	// Error
	E_SA_POS_SM_STATE.ERROR:
		IF ch_ctrl.nCmd = E_SA_CH_CMD.CALIB	THEN
			ch_ctrl.nCmd 			:= E_SA_CH_CMD.NONE;	// Reset command
			stat.nPosState 		:= E_SA_POS_SM_STATE.CALIB;
			stat.bInitialised	:= FALSE;
			stat.sStatus		:= 'Calibrating...';
			M_SetState(E_SA_POS_ELT_STATE.NOTOP);
			M_SetSubstate(E_SA_POS_ELT_SUBSTATE.NOTOP_NOTREADY);
			M_SetNextPosState	:= TRUE;	// State HAS changed
		ELSIF ch_ctrl.nCmd = E_SA_CH_CMD.REF	THEN
			ch_ctrl.nCmd 			:= E_SA_CH_CMD.NONE;	// Reset command
			stat.nPosState 		:= E_SA_POS_SM_STATE.INIT;
			stat.bInitialised	:= FALSE;
			stat.sStatus		:= 'Referencing/INIT Started';
			M_SetState(E_SA_POS_ELT_STATE.NOTOP);
			M_SetSubstate(E_SA_POS_ELT_SUBSTATE.NOTOP_NOTREADY);
			M_SetNextPosState	:= TRUE;	// State HAS changed
		ELSIF ch_ctrl.nCmd = E_SA_CH_CMD.MOV	THEN
			ch_ctrl.nCmd 			:= E_SA_CH_CMD.NONE;	// Reset command
			stat.stState.bACTIVELY_MOVING	:= TRUE;
			stat.stState.bIN_POSITION		:= FALSE;
			stat.nPosState 		:= E_SA_POS_SM_STATE.MOVING;
			stat.nLastPosState 	:= E_SA_POS_SM_STATE.OP;
			stat.sStatus		:= 'Moving...';
			M_SetSubstate(E_SA_POS_ELT_SUBSTATE.OP_MOVING);
			M_SetNextPosState	:= TRUE;	// State HAS changed
		ELSIF ch_ctrl.nCmd = E_SA_CH_CMD.RESET	THEN
			ch_ctrl.nCmd 			:= E_SA_CH_CMD.NONE;	// Reset command
			stat.nPosState 		:= E_SA_POS_SM_STATE.NOT_READY;
			stat.bInitialised	:= FALSE;
			//stat.nErrorCode		:= E_SA_CH_ERROR.OK;
			stat.nErrorCode		:= E_SM_ERROR.OK; 
			stat.sErrorText		:= 'OK';
			stat.sStatus		:= 'Positioner Reset';
			M_SetState(E_SA_POS_ELT_STATE.NOTOP);
			M_SetSubstate(E_SA_POS_ELT_SUBSTATE.NOTOP_NOTREADY);
			M_SetNextPosState	:= TRUE;	// State HAS changed
		ELSE
			stat.sStatus		:= M_GetErrorString();
			M_SetNextPosState	:= FALSE;	// State has NOT changed
		END_IF
END_CASE

*)
END_METHOD

METHOD M_SetState
VAR_INPUT
	nState: E_SA_POS_ELT_STATE;
	//nState: E_RS_BASE_STATE;
END_VAR
stat.nState	:= nState;

// Set substate string
CASE nState	OF
	E_SA_POS_ELT_STATE.NOTOP: 	stat.sState	:= 'NOT OP';
	E_SA_POS_ELT_STATE.OP: 		stat.sState	:= 'OPERATIONAL';
END_CASE
END_METHOD

METHOD M_SetSubstate
VAR_INPUT
	nSubstate: E_SA_POS_ELT_SUBSTATE;
	//nSubstate: E_RS_BASE_SUBSTATE;
END_VAR
stat.nSubstate	:= nSubstate;

// Set substate string
CASE nSubstate	OF
	E_SA_POS_ELT_SUBSTATE.NOTOP_NOTREADY: 		
		stat.sSubstate	:= 'NOT READY';
		stat.sStatus	:= '';
	E_SA_POS_ELT_SUBSTATE.NOTOP_READY: 			stat.sSubstate	:= 'READY';
	E_SA_POS_ELT_SUBSTATE.NOTOP_INITIALIZING:	stat.sSubstate	:= 'INITIALIZING';
	E_SA_POS_ELT_SUBSTATE.NOTOP_ABORTING:		stat.sSubstate	:= 'ABORTING';
	E_SA_POS_ELT_SUBSTATE.NOTOP_ERROR:			stat.sSubstate	:= 'ERROR';
	
	E_SA_POS_ELT_SUBSTATE.OP_STANDSTILL:		stat.sSubstate	:= 'STANDSTILL';            
	E_SA_POS_ELT_SUBSTATE.OP_MOVING:			stat.sSubstate	:= 'MOVING';
	E_SA_POS_ELT_SUBSTATE.OP_SETTING_POS:		stat.sSubstate	:= 'SETTING POS';
	E_SA_POS_ELT_SUBSTATE.OP_STOPPING:			stat.sSubstate	:= 'STOPPING';
	E_SA_POS_ELT_SUBSTATE.OP_ERROR:				stat.sSubstate	:= 'ERROR';
	
END_CASE
END_METHOD

//
// Convert Positioner status from Device to User mode.
//
METHOD M_UpdateStatus
VAR_INPUT
END_VAR
//
// Update bEnabled flag.
// If TRUE, it means that the amplifier is enabled and the sensor is present.
//
//stat.bEnabled	:= stat.stState.bAMPLIFIER_ENABLED AND  stat.stState.bSENSOR_PRESENT;


//
// Set the in-position flag
//
//stat.bInPosition	:= stat.stState.bIN_POSITION;


//
// Set target and actual positions in [UU]
//

//stat.lrPosTarget	:= M_ConvertPosDev2User(stat.devStatus.lnPosTarget);
//stat.lrPosActual	:= M_ConvertPosDev2User(stat.devStatus.lnPosActual);


//
// Set Standard ELT States and Substates
//


//
// Substate
//
CASE stat.nState OF
	E_SA_POS_ELT_STATE.NOTOP:
	/////////////////////////
	IF stat.bError	THEN
		M_SetSubstate(E_SA_POS_ELT_SUBSTATE.NOTOP_ERROR);
	ELSIF	stat.nPosState = E_SA_POS_SM_STATE.NOT_READY	THEN
		M_SetSubstate(E_SA_POS_ELT_SUBSTATE.NOTOP_NOTREADY);
	ELSIF 	stat.nPosState = E_SA_POS_SM_STATE.CALIB  		OR
			stat.nPosState = E_SA_POS_SM_STATE.INIT  		OR
			stat.nPosState = E_SA_POS_SM_STATE.POST_INIT	OR	
			stat.nPosState = E_SA_POS_SM_STATE.CALIB_REF  		THEN
		M_SetSubstate(E_SA_POS_ELT_SUBSTATE.NOTOP_INITIALIZING);
	ELSIF 	stat.nPosState = E_SA_POS_SM_STATE.READY  	THEN
		M_SetSubstate(E_SA_POS_ELT_SUBSTATE.NOTOP_READY);
	ELSE
		M_SetSubstate(E_SA_POS_ELT_SUBSTATE.NOTOP_NOTREADY);
	END_IF
	
	E_SA_POS_ELT_STATE.OP:
	//////////////////////
	IF stat.stState.bACTIVELY_MOVING	THEN
		IF stat.nPosState = E_SA_POS_SM_STATE.STOP	THEN
			M_SetSubstate(E_SA_POS_ELT_SUBSTATE.OP_STOPPING);
		ELSE
			M_SetSubstate(E_SA_POS_ELT_SUBSTATE.OP_MOVING);
		END_IF
	ELSIF stat.stState.bERROR	THEN
		M_SetSubstate(E_SA_POS_ELT_SUBSTATE.OP_ERROR);
	ELSE
		M_SetSubstate(E_SA_POS_ELT_SUBSTATE.OP_STANDSTILL);
	END_IF
END_CASE
END_METHOD

{attribute 'TcRpcEnable':='1'}
{attribute 'TcRpcEnable'}
METHOD RPC_MoveToFilterPosition : INT
VAR_INPUT
	in_nFilterPos:		DINT;	// 1 - 6
	
END_VAR

// If the SmarAct MCS2 Controller is in error,
// the positioner cannot be controlled.
//IF stat.nCtrlErrorCode <> 0  OR  stat.nCtrlState <> E_RS_BASE_STATE.OP THEN
//	RPC_MoveToFilterPosition	:= M_SetRpcStatus(E_SA_RPC_ERROR.CTRL_ERROR);
//	RETURN;
//END_IF


// RPC calls are not allowed in Local mode.
IF stat.bLocal THEN
	RPC_MoveToFilterPosition	:= M_SetRpcStatus(E_SA_RPC_ERROR.LOCAL);
	RETURN;
// Move Absolute command is accepted only in OP state.
ELSIF	stat.nState <> E_SA_POS_ELT_STATE.OP	THEN
	RPC_MoveToFilterPosition	:= M_SetRpcStatus(E_SA_RPC_ERROR.NOT_OP);
	RETURN;
// The positioner has to be initialised / OP (operational), i.e. already REFerenced.
ELSIF	NOT stat.bInitialised	THEN
	RPC_MoveToFilterPosition	:= M_SetRpcStatus(E_SA_RPC_ERROR.CH_NOT_OP);
	RETURN;

// If SW limits are active, check the limits
ELSIF in_nFilterPos > 6  THEN 	
		RPC_MoveToFilterPosition	:= M_SetRpcStatus(E_SA_RPC_ERROR.SW_LIMIT_UPPER);
		RETURN;
ELSIF in_nFilterPos < 1  THEN 	
		RPC_MoveToFilterPosition	:= M_SetRpcStatus(E_SA_RPC_ERROR.SW_LIMIT_LOWER);
		RETURN;
	
END_IF

// Set command
ch_ctrl.nCmd	:= E_SA_CH_CMD.MOV;
ch_ctrl.lrPos	:= in_nFilterPos;



// Call was successful
RPC_MoveToFilterPosition	:= M_SetRpcStatus(E_SA_RPC_ERROR.OK);
END_METHOD

END_FUNCTION_BLOCK

// ---- GlobalTextList.TcGTLO
TEXTLIST GlobalTextList
  14 = '%.2f'
  229 = '%.4f'
  992 = '%.5f'
  28 = '%.6f'
  860 = '%.7f'
  360 = '%s'
  753 = 'Absolute position used by "MOVE ABS"'
  174 = 'Backlash'
  107 = 'GREEN if initialised'
  963 = 'INIT'
  701 = 'Last Command'
  1168 = 'Offset (REL)'
  1376 = 'Position (ABS)'
  510 = 'Position Difference'
  2351 = 'Relative offset used by "MOVE REL"'
  1111 = 'Speed (Pos)'
  1135 = 'Speed (Vel)'
  1119 = 'Target              Actual'
  960 = 'Target           Actual'
END_TEXTLIST

// ---- VISUs/DL_Servo_1_Config.TcVIS
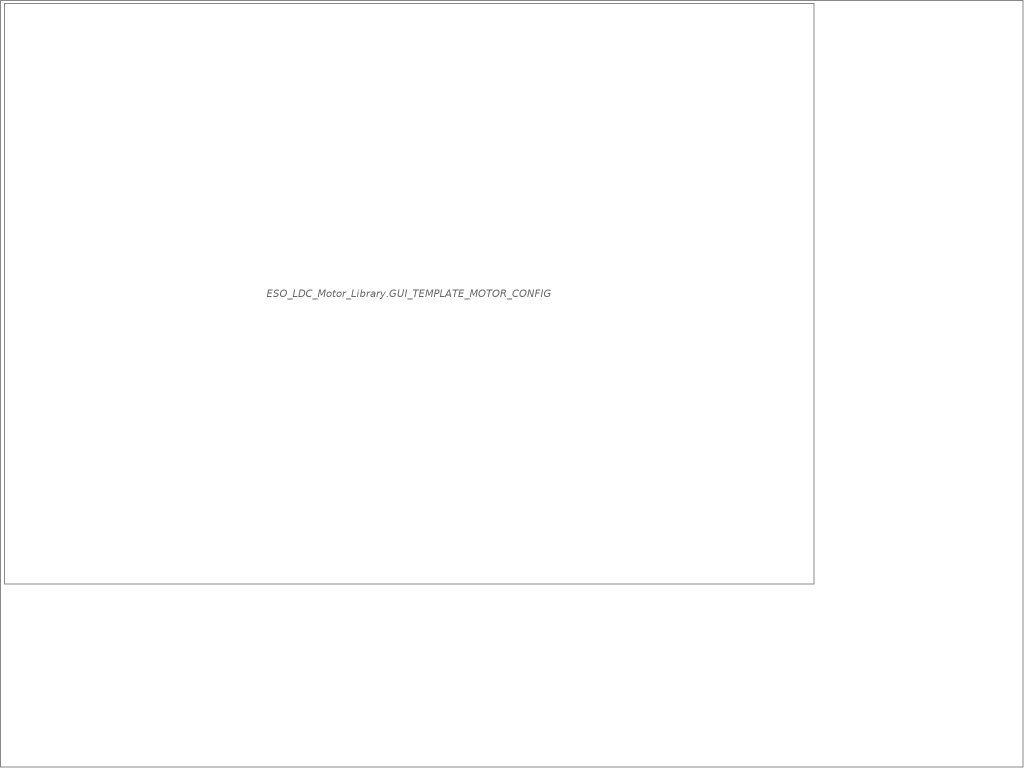
VISUALIZATION DL_Servo_1_Config  // 1024x768
    Frame (4,3 810x581)
        shows ESO_LDC_Motor_Library.GUI_TEMPLATE_MOTOR_CONFIG(m_Instance := MAIN.DL_Servo_1)
END_VISUALIZATION

// ---- VISUs/DL_Servo_1_Control.TcVIS
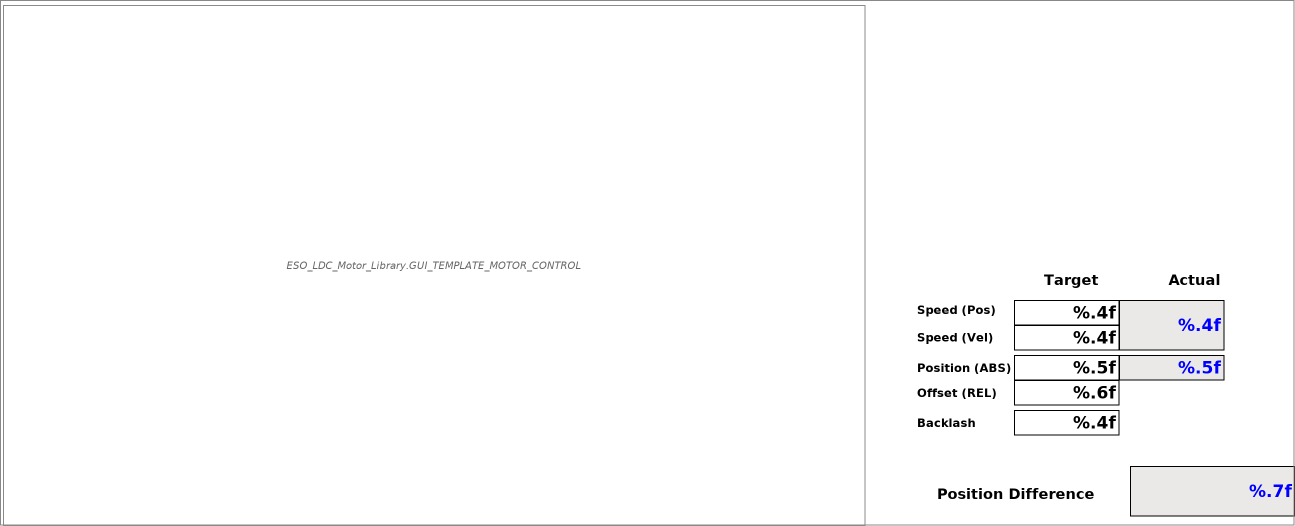
VISUALIZATION DL_Servo_1_Control  // 1295x526
    Frame (3,5 862x521)
        shows ESO_LDC_Motor_Library.GUI_TEMPLATE_MOTOR_CONTROL(m_Instance := MAIN.DL_Servo_1)
    Rectangle (914,300 95x20), "Speed (Pos)"
    Rectangle (1119,355 105x25), "%.5f", text variable: MAIN.DL_Servo_1.stat.lrPosActual, input disabled if: false
    Rectangle (1041,270 190x20), "Target Actual"
    Rectangle (914,358 95x20), "Position (ABS)"
    Rectangle (1119,300 105x50), "%.4f", text variable: MAIN.DL_Servo_1.stat.lrVelActual, input disabled if: false
    Rectangle (1014,325 105x25), "%.4f", text variable: MAIN.DL_Servo_1.ctrl.lrVelocity
        OnMouseDown: write the text variable via Default
    Rectangle (914,413 95x20), "Backlash"
    Rectangle (1014,410 105x25), "%.4f", text variable: MAIN.DL_Servo_1.cfg.lrBacklash
        OnMouseDown: write the text variable via Default
    Rectangle (914,325 95x25), "Speed (Vel)"
    Rectangle (1014,355 105x25), "%.5f", tooltip "Absolute position used by "MOVE ABS"", text variable: MAIN.DL_Servo_1.ctrl.lrPosition
        OnMouseDown: write the text variable via Default
    Rectangle (1014,300 105x25), "%.4f", text variable: MAIN.DL_Servo_1.cfg.lrDefaultVelocity
        OnMouseDown: write the text variable via Default
    Rectangle (914,383 95x20), "Offset (REL)"
    Rectangle (1014,380 105x25), "%.6f", tooltip "Relative offset used by "MOVE REL"", text variable: MAIN.DL_Servo_1.ctrl.lrOffset
        OnMouseDown: write the text variable via Default
    Rectangle (1130,466 165x50), "%.7f", text variable: MAIN.DL_Servo_1.stat.lrPosError, input disabled if: false
    Rectangle (934,484 190x20), "Position Difference"
END_VISUALIZATION

// ---- VISUs/Filter_Wheel.TcVIS
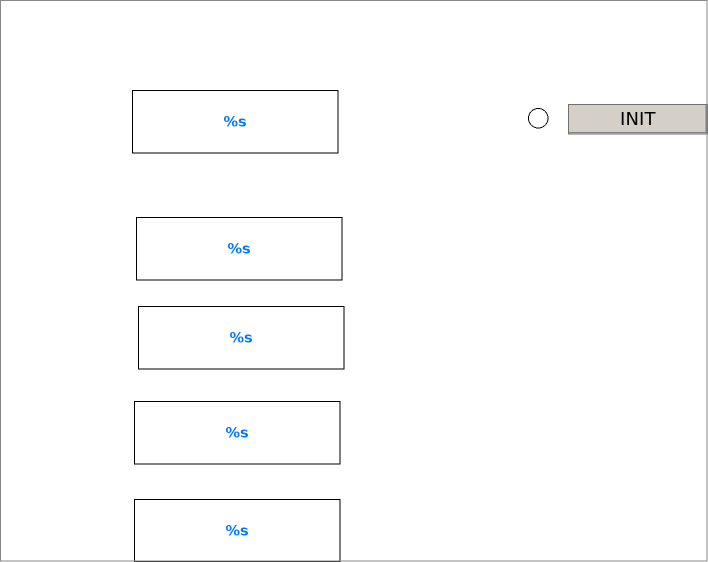
VISUALIZATION Filter_Wheel  // 708x562
    Rectangle (132,90 206x63), "%s", tooltip "Last Command", text variable: MAIN.FILTER_WHEEL.stat.sReply
    Rectangle (136,217 206x63), "%s", tooltip "Last Command", text variable: MAIN.FILTER_WHEEL.stat.sDeviceID
    Rectangle (138,306 206x63), "%s", tooltip "Last Command", text variable: MAIN.FILTER_WHEEL.stat.nCurrentFilterPosition
    Rectangle (134,401 206x63), "%s", tooltip "Last Command", text variable: MAIN.FILTER_WHEEL.stat.sFilterPosition
    Rectangle (134,499 206x63), "%s", tooltip "Last Command", text variable: MAIN.FILTER_WHEEL.stat.bMoveSpeed
    Button (568,104 140x30), "INIT"
        OnMouseClick: execute { MAIN.FILTER_WHEEL.ch_ctrl.nCmd:=E_SA_CH_CMD.REF; }
    Ellipse (528,108 20x20), tooltip "GREEN if initialised", colour toggle: MAIN.FILTER_WHEEL.stat.bInitialised
END_VISUALIZATION

// ---- VISUs/GUI_DL_2.TcVIS
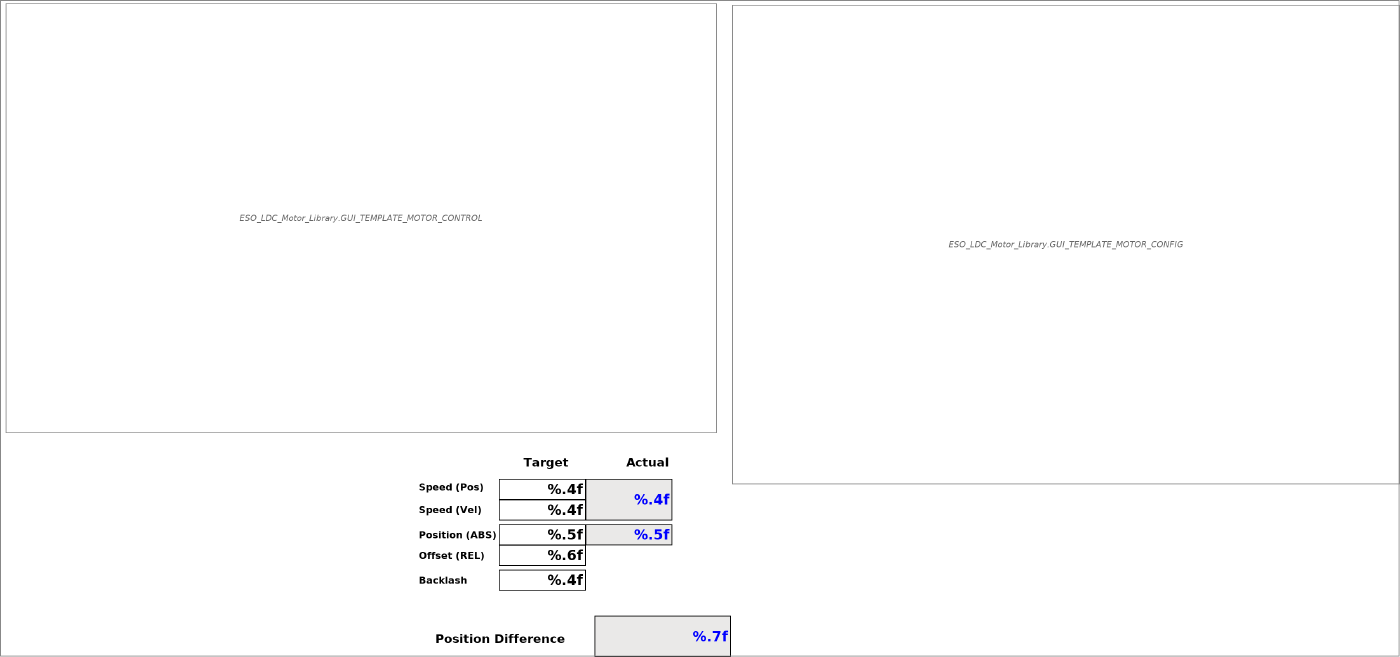
VISUALIZATION GUI_DL_2  // 1698x797
    Frame (7,4 862x521)
        shows ESO_LDC_Motor_Library.GUI_TEMPLATE_MOTOR_CONTROL(m_Instance := MAIN.DL_2)
    Frame (888,6 810x581)
        shows ESO_LDC_Motor_Library.GUI_TEMPLATE_MOTOR_CONFIG(m_Instance := MAIN.DL_2)
    Rectangle (505,581 95x20), "Speed (Pos)"
    Rectangle (710,636 105x25), "%.5f", text variable: MAIN.DL_2.stat.lrPosActual, input disabled if: false
    Rectangle (632,551 190x20), "Target Actual"
    Rectangle (505,639 95x20), "Position (ABS)"
    Rectangle (710,581 105x50), "%.4f", text variable: MAIN.DL_2.stat.lrVelActual, input disabled if: false
    Rectangle (605,606 105x25), "%.4f", text variable: MAIN.DL_2.ctrl.lrVelocity
        OnMouseDown: write the text variable via Default
    Rectangle (505,694 95x20), "Backlash"
    Rectangle (605,691 105x25), "%.4f", text variable: MAIN.DL_2.cfg.lrBacklash
        OnMouseDown: write the text variable via Default
    Rectangle (505,606 95x25), "Speed (Vel)"
    Rectangle (605,636 105x25), "%.5f", tooltip "Absolute position used by "MOVE ABS"", text variable: MAIN.DL_2.ctrl.lrPosition
        OnMouseDown: write the text variable via Default
    Rectangle (605,581 105x25), "%.4f", text variable: MAIN.DL_2.cfg.lrDefaultVelocity
        OnMouseDown: write the text variable via Default
    Rectangle (505,664 95x20), "Offset (REL)"
    Rectangle (605,661 105x25), "%.6f", tooltip "Relative offset used by "MOVE REL"", text variable: MAIN.DL_2.ctrl.lrOffset
        OnMouseDown: write the text variable via Default
    Rectangle (721,747 165x50), "%.7f", text variable: MAIN.DL_2.stat.lrPosError, input disabled if: false
    Rectangle (525,765 190x20), "Position Difference"
END_VISUALIZATION

// ---- VISUs/GUI_TIME_INFORMATION.TcVIS
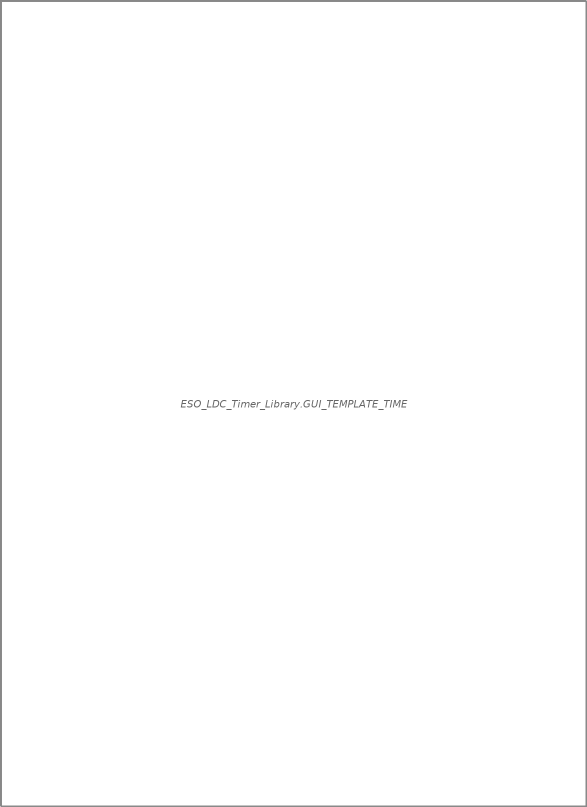
VISUALIZATION GUI_TIME_INFORMATION  // 587x807
    Frame (1,1 586x806)
        shows ESO_LDC_Timer_Library.GUI_TEMPLATE_TIME(m_Instance := MAIN.time_info)
END_VISUALIZATION

// ---- VISUs/Shutter_1.TcVIS
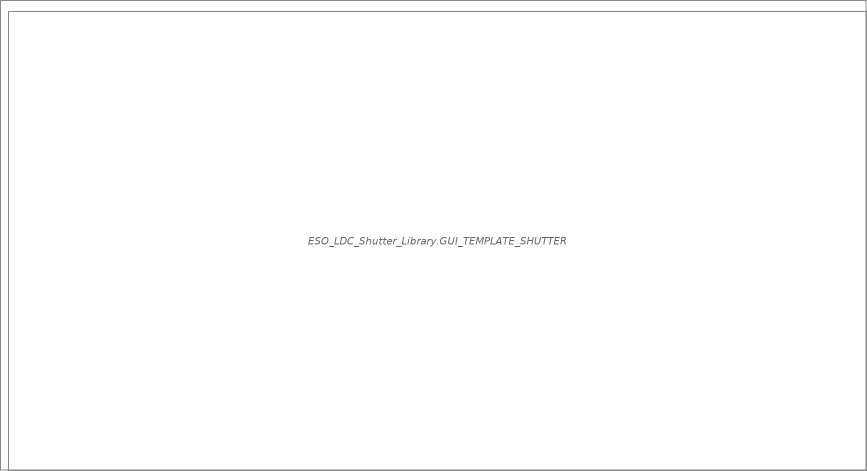
VISUALIZATION Shutter_1  // 867x471
    Frame (8,11 859x460)
        shows ESO_LDC_Shutter_Library.GUI_TEMPLATE_SHUTTER(m_Instance := MAIN.shutter_1)
END_VISUALIZATION

// ---- VISUs/TipTilt_Servo_1.TcVIS
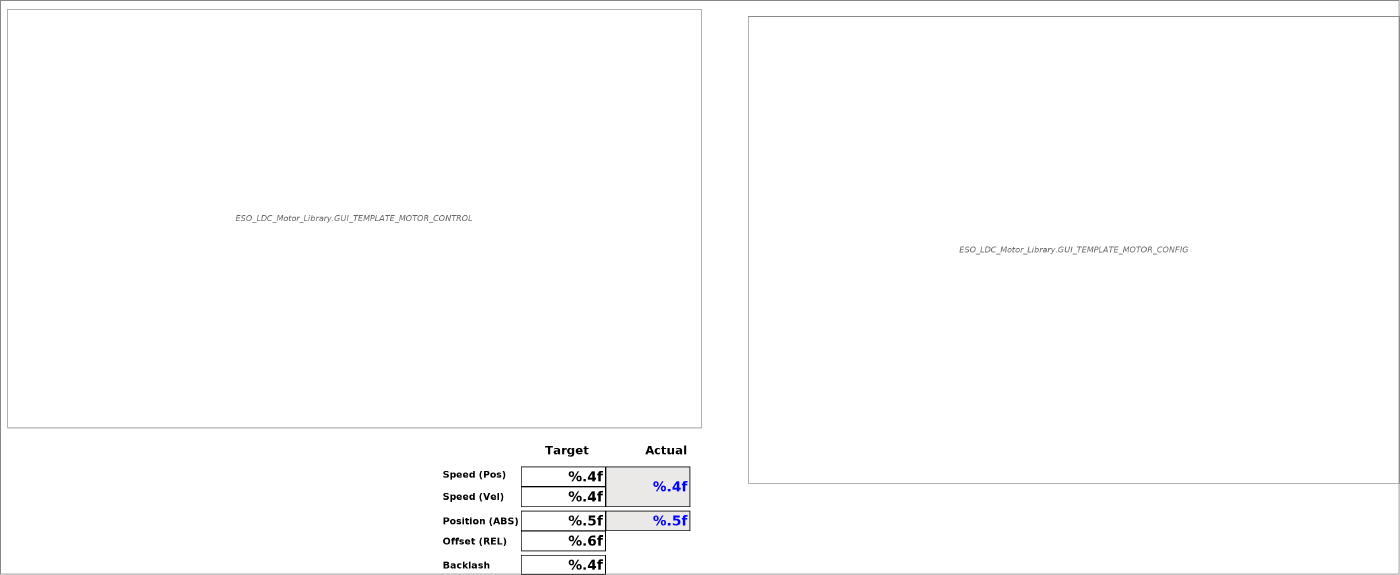
VISUALIZATION TipTilt_Servo_1  // 1739x715
    Frame (9,11 862x521)
        shows ESO_LDC_Motor_Library.GUI_TEMPLATE_MOTOR_CONTROL(m_Instance := MAIN.tiptilt_1)
    Frame (929,20 810x581)
        shows ESO_LDC_Motor_Library.GUI_TEMPLATE_MOTOR_CONFIG(m_Instance := MAIN.tiptilt_1)
    Rectangle (547,580 95x20), "Speed (Pos)"
    Rectangle (752,635 105x25), "%.5f", text variable: MAIN.tiptilt_1.stat.lrPosActual, input disabled if: false
    Rectangle (674,550 190x20), "Target Actual"
    Rectangle (547,638 95x20), "Position (ABS)"
    Rectangle (752,580 105x50), "%.4f", text variable: MAIN.tiptilt_1.stat.lrVelActual, input disabled if: false
    Rectangle (647,605 105x25), "%.4f", text variable: MAIN.tiptilt_1.ctrl.lrVelocity
        OnMouseDown: write the text variable via Default
    Rectangle (547,693 95x20), "Backlash"
    Rectangle (647,690 105x25), "%.4f", text variable: MAIN.tiptilt_1.cfg.lrBacklash
        OnMouseDown: write the text variable via Default
    Rectangle (547,605 95x25), "Speed (Vel)"
    Rectangle (647,635 105x25), "%.5f", tooltip "Absolute position used by "MOVE ABS"", text variable: MAIN.tiptilt_1.ctrl.lrPosition
        OnMouseDown: write the text variable via Default
    Rectangle (647,580 105x25), "%.4f", text variable: MAIN.tiptilt_1.cfg.lrDefaultVelocity
        OnMouseDown: write the text variable via Default
    Rectangle (547,663 95x20), "Offset (REL)"
    Rectangle (647,660 105x25), "%.6f", tooltip "Relative offset used by "MOVE REL"", text variable: MAIN.tiptilt_1.ctrl.lrOffset
        OnMouseDown: write the text variable via Default
END_VISUALIZATION
